(* CODESYS project Dbg.library
   Company: _
   DefaultNamespace: Debug
   Title: Debug
   Placeholder: _Debug
   Author: Krystian Lis et al.
   Description: Code debugging helper.
   Version: 1.0.0

Project tree, tasks and I/O mapping:
  libraries: Strings, * (_)
  Dbg/
    global variables _Debug
    function DebugLen [ST]
    function block DebugList [ST]
    function DebugMsg [ST]
    interface I_Debug
    global variables Param
    data type ST_DebugInfo
*)

// Dbg/ST_DebugInfo
TYPE INTERNAL ST_DebugInfo :
STRUCT
	iDebug		: I_Debug;
	sInfo		: Strings.Str;
END_STRUCT
END_TYPE

// Dbg/_Debug
{attribute 'qualified_only'}
VAR_GLOBAL INTERNAL
	stDebug				: ARRAY[0..Param.nMaxDebugArraySize] OF ST_DebugInfo;
	nDebugLen			: UDINT;	
END_VAR

// Dbg/Param
{attribute 'qualified_only'}
VAR_GLOBAL CONSTANT
	nMaxDebugArraySize		: UDINT := 10;
END_VAR

// Dbg/DebugLen
FUNCTION DebugLen : UDINT

DebugLen := _Debug.nDebugLen;

END_FUNCTION

// Dbg/DebugList
FUNCTION_BLOCK DebugList
VAR
	_refDebug			: REFERENCE TO ARRAY[0..Param.nMaxDebugArraySize] OF ST_DebugInfo REF= _Debug.stDebug;
END_VAR

END_FUNCTION_BLOCK

// Dbg/DebugMsg
FUNCTION DebugMsg
VAR_INPUT
	iDebug			: I_Debug;
	sInfo			: Strings.Str;
END_VAR
VAR
END_VAR

IF _Debug.nDebugLen = Param.nMaxDebugArraySize THEN
	RETURN;	
ELSIF _Debug.nDebugLen = Param.nMaxDebugArraySize - 1 THEN
	_Debug.stDebug[_Debug.nDebugLen].iDebug := 0;
	_Debug.stDebug[_Debug.nDebugLen].sInfo := 'Debug overflow!';
	RETURN;
END_IF

_Debug.stDebug[_Debug.nDebugLen].iDebug := iDebug;
_Debug.stDebug[_Debug.nDebugLen].sInfo := sInfo;
_Debug.nDebugLen := _Debug.nDebugLen + 1;

END_FUNCTION

// Dbg/I_Debug
INTERFACE I_Debug

END_INTERFACE
